PROGRAM EndLogic
VAR
	fbRTRIG: R_TRIG;
	fbRTRIGFillInUpper : R_TRIG;
END_VAR
VAR_INPUT
//	In : INT;
	nCurrentBlock: BOOL;
END_VAR
VAR_OUTPUT
	OutputBool : BOOL;
END_VAR



fbRTRIG(CLK:=nCurrentBlock , Q=> ); 

OutputBool := fbRTRIG.Q;

END_PROGRAM

(* stored: Version 1.1.0.1, ProductVersion 3.1.4024.5
   POU EndLogic: Id {71e1561f-8207-47a3-99b7-aa8be5bb6b09}, SpecialFunc None *)
